{attribute 'qualified_only'}
TYPE ENUM_XPIM_States :
(
    Unknown := 0,
    OUT := 1,
    YAG := 2,
    DIAMOND := 3,
    RETICLE := 4
);
END_TYPE

(* stored: Version 1.1.0.1, ProductVersion 3.1.4022.18
   DUT ENUM_XPIM_States: Id {f0241cec-71d0-42c5-9fc1-9ae15c8cbd48} *)
